// TIA Portal V20 export
// export: Created 2026-04-11T06:02:30.2660084Z, ExportSetting WithDefaults, DisplayName Totally Integrated Automation Portal, DisplayVersion V20, DisplayName TIA Portal Openness, DisplayVersion V20, DisplayName TIA Portal Version Control Interface, DisplayVersion V20, DisplayName STEP 7 Professional, DisplayVersion V20, DisplayName STEP 7 Safety, DisplayVersion V20, DisplayName WinCC Basic/Comfort/Advanced, DisplayVersion V20, DisplayName WinCC Unified, DisplayVersion V20
TYPE "udtHMI_AnalogInput"
// stored: IsFailsafeCompliant false
   STRUCT
      iMode : Int;   // Current mode
      iErrorCode { ExternalWritable := 'False'} : Int;   // Error code
      iStatus { ExternalWritable := 'False'} : Int;   // Overall HMI Status
      rActiveValue { ExternalWritable := 'False'} : Real;   // Used Value, Input or Override
      rInputValue { ExternalWritable := 'False'} : Real;   // Input Value
      rManualValue { S7_SetPoint := 'True'} : Real;   // Manual mode simulated value
      bPB_ResetError : Bool;   // PB Reset block errors
      bPBEN_ResetError { ExternalWritable := 'False'} : Bool;   // PB Reset error enabled
      bError { ExternalWritable := 'False'} : Bool;   // Overall error
   END_STRUCT;
END_TYPE
